// TwinCAT 3 PLC project PLC1
// ProgramVersion: 3.1.4024.0
// libraries:
//   Tc2_Standard, * (Beckhoff Automation GmbH)
//   Tc2_System, * (Beckhoff Automation GmbH)
//   Tc3_Module, * (Beckhoff Automation GmbH)
// project tree:
//   / PlcTask.TcTTO
//   POUs/ FB_Clock.TcPOU (not stored), MAIN.TcPOU
// real-time tasks:
//   TASK PlcTask: cycle T#10ms, priority 20, ADS port 350

CONFIGURATION PLC1
    RESOURCE PLC ON TwinCAT3
        TASK PlcTask(INTERVAL := T#10ms, PRIORITY := 20);
        PROGRAM MAIN WITH PlcTask : MAIN;
    END_RESOURCE
END_CONFIGURATION

// ---- POUs/MAIN.TcPOU
PROGRAM MAIN
VAR
	fbClockOneSecond : FB_CLOCK;
	fbClock250ms	 : FB_CLOCK;
	fbClock500ms 	 : FB_CLOCK;
END_VAR

fbClockOneSecond(TIME_ON:=T#500MS, TIME_OFF:=T#500MS, OUT_CLK=>);
fbClock250ms(TIME_ON:=T#125MS, TIME_OFF:=T#125MS, OUT_CLK=>);
fbClock500ms(TIME_ON:=T#250MS, TIME_OFF:=T#250MS, OUT_CLK=>);

END_PROGRAM
